FUNCTION_BLOCK MockDeserializableUserObject IMPLEMENTS I_Deserializable
VAR
	_name : STRING;
	_age : INT;
END_VAR

PROPERTY PUBLIC Age : INT
GET
Age := _age;
END_GET
SET
_age := Age;
END_SET
END_PROPERTY

METHOD PRIVATE CreateMissingKeyError : I_Error
VAR_INPUT
END_VAR
END_METHOD

PROPERTY PUBLIC Name : STRING
GET
Name := _name;
END_GET
SET
_name := Name;
END_SET
END_PROPERTY

METHOD TryDeserializeFrom : BOOL
VAR_INPUT
	Deserializer : I_Deserializer;
	Feedback : I_DeserializerFeedback;
END_VAR
IF NOT Deserializer.TryGetKeyString('Name',_name, Feedback) THEN
	RETURN;
END_IF

IF NOT Deserializer.TryGetKeyInt('Age',_age, Feedback) THEN
	RETURN;
END_IF

TryDeserializeFrom := TRUE;
END_METHOD

END_FUNCTION_BLOCK

(* stored: Version 1.1.0.1, ProductVersion 3.1.4024.12
   POU MockDeserializableUserObject: Id {26a5c0a0-9bcd-4053-ae19-dc4ef45f044f}, SpecialFunc None
   Folder Private: Id {aee6b500-d615-4113-9cf2-7ee1d615d6aa}
   Property Age: Id {75bb5ecc-a1d1-4e89-b4ae-786a501e6734}
   Get Get: Id {41015d26-0512-4db6-8c2d-57dbe1fc5103}
   Set Set: Id {7e3637e1-3186-4a14-9313-0353d41b8722}
   Method CreateMissingKeyError: Id {3a65d5e3-ba4f-40e0-b0f1-732ac1e9f147}
   Property Name: Id {462ded79-a15b-4005-b9f0-06ef83902385}
   Get Get: Id {a5665efe-bd30-4fe7-88d7-edfcfda2ac11}
   Set Set: Id {bdda4c86-0c39-4b25-9ae7-863ff8453a8a}
   Method TryDeserializeFrom: Id {d6e880b1-1bdb-47e0-b960-89d475fdcf1a} *)
